  rq_wait_ft_sensor_steady(2000)
  zero_ftsensor()
  sleep(0.1)
  # end: URCap Program Node
  # begin: URCap Program Node
  #   Source: Robotiq_Copilot, 1.22.1.14215, Robotiq Inc.
  #   Type: Find Surface
  $ 62 "Find Surface"
  zero_ftsensor()
  sleep(0.1)
  surface_found = rq_linear_search_urcap("Z+", 10.000, 0.005000, 0.100000, 1)
  storevar.setvariablepose("rq_findSurface_8f0967cc-59bf-4555-8a29-6c49c2e47a29_exitPosition", get_actual_tcp_pose())
  $ 63 "'Add Stop conditions from the Find Surface node'" "noBreak"
  # 'Add Stop conditions from the Find Surface node'
  # end: URCap Program Node
  # begin: URCap Program Node
  #   Source: Robotiq_Copilot, 1.22.1.14215, Robotiq Inc.
  #   Type: Finishing Tool Control
  $ 64 "Start tool"
  set_standard_digital_out(0, True)
  # end: URCap Program Node
  $ 65 "Wait: 0.5"
  sleep(0.5)
  $ 66 "Force"
  sleep(0.02)
  zero_ftsensor()
  force_mode(tool_pose(), [0, 0, 1, 0, 0, 0], [0.0, 0.0, 1.0, 0.0, 0.0, 0.0], 2, [0.1, 0.1, 0.15, 0.3490658503988659, 0.3490658503988659, 0.3490658503988659])
  $ 67 "Waypoint_7" "noBreak"
  set_tcp(p[0.00318,0.11464,0.09820000000000001,-0.7853981633974483,0.0,0.0])
  movel(pose_trans(CubeFront, pose_trans(p[-.005597006121, -.192408094989, .653246871754, -1.571622694982, -.002967386491, .002471774867], Waypoint_7_p)), a=1.2, v=0.05)
  end_force_mode()
  stopl(5.0)
  # begin: URCap Program Node
  #   Source: Robotiq_Copilot, 1.22.1.14215, Robotiq Inc.
  #   Type: Finishing Tool Control
  $ 68 "Stop tool"
  set_standard_digital_out(0, False)
  # end: URCap Program Node
  $ 69 "Waypoint_13" "breakAfter"
  set_tcp(p[0.00318,0.11464,0.09820000000000001,-0.7853981633974483,0.0,0.0])
  movel(pose_trans(CubeFront, pose_trans(p[-.002001169423, -.178123008725, .618090231485, -1.568699287997, .013964727372, .007428573496], Waypoint_13_p)), a=1.2, v=0.25)
  $ 70 "Waypoint_9" "breakAfter"
  set_tcp(p[0.00318,0.11464,0.09820000000000001,-0.7853981633974483,0.0,0.0])
  movel(pose_trans(CubeFront, pose_trans(p[-.002001169423, -.178123008725, .618090231485, -1.568699287997, .013964727372, .007428573496], Waypoint_9_p)), a=1.2, v=0.25)
  $ 71 "clear" "breakAfter"
  set_tcp(p[0.00318,0.11464,0.09820000000000001,-0.7853981633974483,0.0,0.0])
  movel(pose_trans(CubeFront, pose_trans(p[-.002001169423, -.178123008725, .618090231485, -1.568699287997, .013964727372, .007428573496], clear_p)), a=1.2, v=0.25)
  $ 104 "SprayFront"
  $ 105 "MoveJ"
  $ 106 "clear" "breakAfter"
  set_tcp(p[0.00318,0.11464,0.09820000000000001,-0.7853981633974483,0.0,0.0])
  movej(get_inverse_kin(pose_trans(CubeFront, pose_trans(p[-.002001169423, -.178123008725, .618090231485, -1.568699287997, .013964727372, .007428573496], clear_p)), qnear=clear_q), a=1.3962634015954636, v=1.0471975511965976)
  $ 107 "MoveJ"
  $ 108 "Waypoint_10" "breakAfter"
  set_tcp(p[0.020839023181949995,-0.027139950822234082,0.10599373590389219,0.12258870209179472,1.1769383890382668,2.869747076630172])
  movej(get_inverse_kin(pose_trans(CubeFront, pose_trans(p[-.002001169423, -.178123008725, .618090231485, -1.568699287997, .013964727372, .007428573496], Waypoint_10_p)), qnear=Waypoint_10_q), a=1.3962634015954636, v=1.0471975511965976)
  $ 109 "Call StartSpray"
  StartSpray()
  $ 110 "MoveL"
  $ 111 "Waypoint_12" "breakAfter"
  movel(pose_trans(CubeFront, pose_trans(p[-.002001169423, -.178123008725, .618090231485, -1.568699287997, .013964727372, .007428573496], Waypoint_12_p)), a=1.2, v=0.1)
  $ 112 "Call stopSpray"
  stopSpray()
  $ 113 "MoveJ"
  $ 114 "Waypoint_21" "breakAfter"
  set_tcp(p[0.020839023181949995,-0.027139950822234082,0.10599373590389219,0.12258870209179472,1.1769383890382668,2.869747076630172])
  movej(get_inverse_kin(pose_trans(CubeFront, pose_trans(p[-.002001169423, -.178123008725, .618090231485, -1.568699287997, .013964727372, .007428573496], Waypoint_21_p)), qnear=Waypoint_21_q), a=1.3962634015954636, v=1.0471975511965976)
  $ 115 "Call StartSpray"
  StartSpray()
  $ 116 "MoveL"
  $ 117 "Waypoint_22" "breakAfter"
  set_tcp(p[0.020839023181949995,-0.027139950822234082,0.10599373590389219,0.12258870209179472,1.1769383890382668,2.869747076630172])
  movel(pose_trans(CubeFront, pose_trans(p[-.002001169423, -.178123008725, .618090231485, -1.568699287997, .013964727372, .007428573496], Waypoint_22_p)), a=1.2, v=0.1)
  $ 118 "Call stopSpray"
  stopSpray()
  $ 119 "MoveJ"
  $ 120 "Waypoint_23" "breakAfter"
  set_tcp(p[0.020839023181949995,-0.027139950822234082,0.10599373590389219,0.12258870209179472,1.1769383890382668,2.869747076630172])
  movej(get_inverse_kin(pose_trans(CubeFront, pose_trans(p[-.002001169423, -.178123008725, .618090231485, -1.568699287997, .013964727372, .007428573496], Waypoint_23_p)), qnear=Waypoint_23_q), a=1.3962634015954636, v=1.0471975511965976)
  $ 121 "Call StartSpray"
  StartSpray()
  $ 122 "MoveL"
  $ 123 "Waypoint_24" "breakAfter"
  set_tcp(p[0.020839023181949995,-0.027139950822234082,0.10599373590389219,0.12258870209179472,1.1769383890382668,2.869747076630172])
  movel(pose_trans(CubeFront, pose_trans(p[-.002001169423, -.178123008725, .618090231485, -1.568699287997, .013964727372, .007428573496], Waypoint_24_p)), a=1.2, v=0.1)
  $ 124 "Call stopSpray"
  stopSpray()
  $ 125 "MoveJ"
  $ 126 "clear" "breakAfter"
  movej(clear_q, a=1.3962634015954636, v=1.0471975511965976)
  $ 127 "MoveJ"
  $ 128 "Waypoint_26" "breakAfter"
  set_tcp(p[0.020839023181949995,-0.027139950822234082,0.10599373590389219,0.12258870209179472,1.1769383890382668,2.869747076630172])
  movej(get_inverse_kin(pose_trans(CubeFront, pose_trans(p[-.002001169423, -.178123008725, .618090231485, -1.568699287997, .013964727372, .007428573496], Waypoint_26_p)), qnear=Waypoint_26_q), a=1.3962634015954636, v=1.0471975511965976)
  $ 129 "Call StartSpray"
  StartSpray()
  $ 130 "MoveL"
  $ 131 "Waypoint_25" "breakAfter"
  set_tcp(p[0.020839023181949995,-0.027139950822234082,0.10599373590389219,0.12258870209179472,1.1769383890382668,2.869747076630172])
  movel(pose_trans(CubeFront, pose_trans(p[-.002001169423, -.178123008725, .618090231485, -1.568699287997, .013964727372, .007428573496], Waypoint_25_p)), a=1.2, v=0.1)
  $ 132 "Call stopSpray"
  stopSpray()
  $ 133 "MoveJ"
  $ 134 "clear" "breakAfter"
  movej(clear_q, a=1.3962634015954636, v=1.0471975511965976)
  $ 135 "SprayRebate"
  $ 136 "MoveJ"
  $ 137 "clear" "breakAfter"
  movej(clear_q, a=1.3962634015954636, v=1.0471975511965976)
  $ 138 "MoveJ"
  $ 139 "Waypoint_28" "breakAfter"
  set_tcp(p[0.020839023181949995,-0.027139950822234082,0.10599373590389219,0.12258870209179472,1.1769383890382668,2.869747076630172])
  movej(get_inverse_kin(pose_trans(CubeFront, pose_trans(p[-.002001169423, -.178123008725, .618090231485, -1.568699287997, .013964727372, .007428573496], Waypoint_28_p)), qnear=Waypoint_28_q), a=1.3962634015954636, v=1.0471975511965976)
  $ 140 "Call StartSpray"
  StartSpray()
  $ 141 "MoveL"
  $ 142 "Waypoint_27" "breakAfter"
  set_tcp(p[0.020839023181949995,-0.027139950822234082,0.10599373590389219,0.12258870209179472,1.1769383890382668,2.869747076630172])
  movel(pose_trans(CubeFront, pose_trans(p[-.002001169423, -.178123008725, .618090231485, -1.568699287997, .013964727372, .007428573496], Waypoint_27_p)), a=1.2, v=0.1)
  $ 143 "Call stopSpray"
  stopSpray()
  $ 144 "MoveJ"
  $ 145 "Waypoint_29" "breakAfter"
  set_tcp(p[0.020839023181949995,-0.027139950822234082,0.10599373590389219,0.12258870209179472,1.1769383890382668,2.869747076630172])
  movej(get_inverse_kin(pose_trans(CubeFront, pose_trans(p[-.002001169423, -.178123008725, .618090231485, -1.568699287997, .013964727372, .007428573496], Waypoint_29_p)), qnear=Waypoint_29_q), a=1.3962634015954636, v=1.0471975511965976)
  $ 146 "Call StartSpray"
  StartSpray()
  $ 147 "MoveL"
  $ 148 "Waypoint_30" "breakAfter"
  set_tcp(p[0.020839023181949995,-0.027139950822234082,0.10599373590389219,0.12258870209179472,1.1769383890382668,2.869747076630172])
  movel(pose_trans(CubeFront, pose_trans(p[-.002001169423, -.178123008725, .618090231485, -1.568699287997, .013964727372, .007428573496], Waypoint_30_p)), a=1.2, v=0.1)
  $ 149 "Call stopSpray"
  stopSpray()
  $ 150 "MoveJ"
  $ 151 "clear" "breakAfter"
  movej(clear_q, a=1.3962634015954636, v=1.0471975511965976)
  $ 152 "MoveJ"
  $ 153 "Waypoint_32" "breakAfter"
  set_tcp(p[0.020839023181949995,-0.027139950822234082,0.10599373590389219,0.12258870209179472,1.1769383890382668,2.869747076630172])
  movej(get_inverse_kin(pose_trans(CubeFront, pose_trans(p[-.002001169423, -.178123008725, .618090231485, -1.568699287997, .013964727372, .007428573496], Waypoint_32_p)), qnear=Waypoint_32_q), a=1.3962634015954636, v=1.0471975511965976)
  $ 154 "Call StartSpray"
  StartSpray()
  $ 155 "MoveL"
  $ 156 "Waypoint_33" "breakAfter"
  set_tcp(p[0.020839023181949995,-0.027139950822234082,0.10599373590389219,0.12258870209179472,1.1769383890382668,2.869747076630172])
  movel(pose_trans(CubeFront, pose_trans(p[-.002001169423, -.178123008725, .618090231485, -1.568699287997, .013964727372, .007428573496], Waypoint_33_p)), a=1.2, v=0.1)
  $ 157 "Call stopSpray"
  stopSpray()
  $ 158 "MoveJ"
  $ 159 "clear" "breakAfter"
  movej(clear_q, a=1.3962634015954636, v=1.0471975511965976)
end
